{attribute 'qualified_only'}
{attribute 'strict'}
TYPE eGuidanceSystemSTM :
(
	Initializing,
	PreRunning,
	Running,
	PostRunning
);
END_TYPE

(* stored: Version 1.1.0.1, ProductVersion 3.1.4024.12
   DUT eGuidanceSystemSTM: Id {2ca63699-51e4-48fd-999a-7300694d43a0} *)
